FUNCTION_BLOCK B_TRIG
VAR_INPUT
	CLK : BOOL;
END_VAR
VAR_OUTPUT
	Q : BOOL;
END_VAR
VAR
	edge : BOOL;
END_VAR

(*
version 1.0	4. aug. 2006
programmer 	hugo
tested by		tobias

this block is similar to R_trig and F_trig but it generates a pulse on rising and falling edge.

*)

Q := clk XOR edge;
edge := CLK;


(* revision history
hm		4. aug. 2006	rev 1.0
	original version

*)

END_FUNCTION_BLOCK

(* stored: Version 1.1.0.1, ProductVersion 3.1.4022.7
   POU B_TRIG: Id {8df87104-1c06-4b8a-87a8-c7b3bcb67805}, SpecialFunc None *)
